// TIA Portal V19 export
FUNCTION "CONTROL BALANCE TANK" : Void   // FC24, STL
TITLE = CONTROL LEVEL CIP TANK
{ S7_Optimized_Access := 'TRUE' }
NAME : CIPTANK
VERSION : 0.0
// Comment
// stored: AutoNumber false
BEGIN

NETWORK
TITLE = CONTROL LEVEL CIP TANK
// Comment
      AN    "TANK AUTO";
      AN    "CONTROL CIP TANK";
      R     "MY0115";
      BEC;
      A     "B01.41";
      R     "MY0115";
      BEC;
      AN    "B01.42";
      S     "MY0115";
      NOP   0;
END_FUNCTION
